Staubli VAL3: connectHostRos.dtx

mdesc mNomSpeed
public sio soTcpIpFbk
public sio siTcpIpMotion
public num nRecvData[53]
public CommParameter cRosMotionParm
  [0]
    num port
    string target
    num clients
    num endOfString
    num timeOut
    num baudRate
    string parity
    num bits
    num stopBits
    string mode
    string flowControl
    bool nagle
public CommParameter cRosFbkParm
  [0]
    num port
    string target
    num clients
    num endOfString
    num timeOut
    num baudRate
    string parity
    num bits
    num stopBits
    string mode
    string flowControl
    bool nagle
public FlagStatus fRosStatus
  [0]
    num ForceFlag
    num RosFlag
    num RobotFlag
public num nSendData[52]
